ABB RobotStudio station: palet.rspag

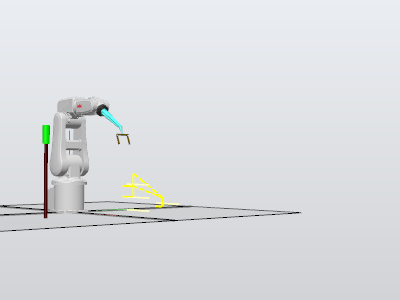
--- station ---
Station palet (saved by RobotStudio 25.3.11371.0)
Controller IRB120_3_58
  mechanical unit ROB_1: IRB120_3_58__01, 6 joints, base frame (0, 0, 0) mm
Layout (positions relative to the parent item):
  - IRB120_3_58__01 [mechanism, from %ABB.RobotStudio.Models.IRB120%\IRB120_3_58_G_01.rslib] at (0, 0, 0) mm; joint values [0, 0, 0, 0, 0.5236, 0] (rad or m)
  - traspalet [mechanism] at (364.35, 0, 594) mm, rotated rx 180 ry 60 rz 180 deg
      TCP traspalet at (31.79, 0, 229.64) mm, rotated rx 0 ry 38 rz 0 deg
      links: mytool3palet
  - YOGUR [smart component]
      signals: DI borra
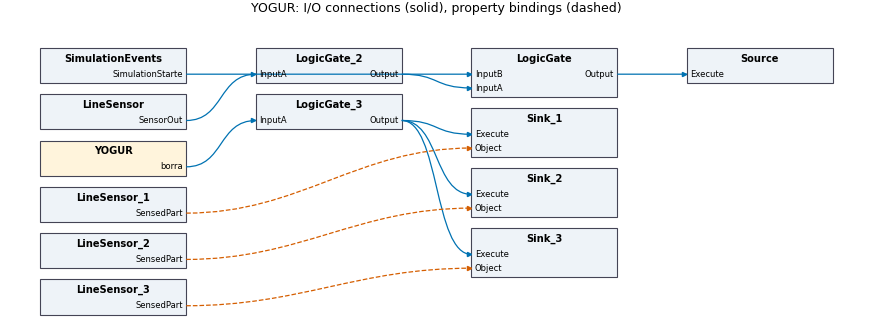
      connections:
        SimulationEvents.SimulationStarted -> LogicGate.InputB
        LogicGate.Output -> Source.Execute
        LineSensor.SensorOut -> LogicGate_2.InputA
        LogicGate_2.Output -> LogicGate.InputA
        YOGUR.borra -> LogicGate_3.InputA
        LogicGate_3.Output -> Sink_3.Execute
        LogicGate_3.Output -> Sink_2.Execute
        LogicGate_3.Output -> Sink_1.Execute
        LineSensor_1.SensedPart => Sink_1.Object
        LineSensor_2.SensedPart => Sink_2.Object
        LineSensor_3.SensedPart => Sink_3.Object
    - yogur [part] at (0, 0, 0) mm, size 60 x 80 x 72 mm
    - Source [smart component, from Components\Source.rslib]
        properties: Source=yogur; Copy=(none); Parent=(none); Position=[0.7 0.2 0]; Orientation=[0 0 0]; Transient=true; PhysicsBehavior=-1
    - SimulationEvents [smart component, from Components\SimulationEvents.rslib]
    - LogicGate [smart component, from Components\LogicGate.rslib]
        properties: Operator=OR; Delay=0
    - LineSensor [smart component, from Components\LineSensor.rslib]
        properties: Start=[0.6 0.2 0.07]; End=[0.8 0.2 0.07]; Length=0.2; Radius=0; Tag=(none); SenseMultiple=false; SensedPart=(none); SensedPoint=[0.67 0.2 0.07]
      - _sensorPart_ [part], size 200 x 0 x 0 mm
    - LogicGate_2 [smart component, from Components\LogicGate.rslib]
        properties: Operator=NOT; Delay=1
    - LineSensor_1 [smart component, from Components\LineSensor.rslib]
        properties: Start=[0.6 -0.01 0.04]; End=[0.8 -0.01 0.04]; Length=0.2; Radius=0; Tag=(none); SenseMultiple=false; SensedPart=(none); SensedPoint=[0.675910827636719 -0.00999999904632568 0.0400000038146973]
      - _sensorPart_ [part], size 200 x 0 x 0 mm
    - LineSensor_2 [smart component, from Components\LineSensor.rslib]
        properties: Start=[0.6 -0.01 0.11]; End=[0.8 -0.01 0.11]; Length=0.2; Radius=0; Tag=(none); SenseMultiple=false; SensedPart=(none); SensedPoint=[0.675313598632812 -0.01 0.11]
      - _sensorPart_ [part], size 200 x 0 x 0 mm
    - LineSensor_3 [smart component, from Components\LineSensor.rslib]
        properties: Start=[0.6 -0.01 0.18]; End=[0.8 -0.01 0.18]; Length=0.2; Radius=0; Tag=(none); SenseMultiple=false; SensedPart=(none); SensedPoint=[0 0 0]
      - _sensorPart_ [part], size 200 x 0 x 0 mm
    - Sink_1 [smart component, from Components\Sink.rslib]
        properties: Object=(none)
    - Sink_3 [smart component, from Components\Sink.rslib]
        properties: Object=(none)
    - Sink_2 [smart component, from Components\Sink.rslib]
        properties: Object=(none)
    - LogicGate_3 [smart component, from Components\LogicGate.rslib]
        properties: Operator=NOT; Delay=0
  - BALIZA [smart component]
      signals: DI COLOR
      connections:
        BALIZA.COLOR -> Highlighter.Active
    - BALIZA [part] at (400, -400, 0) mm, size 40 x 39.9 x 100 mm
    - Highlighter [smart component, from Components\Highlighter.rslib]
        properties: Object=BALIZA; Color=[255 0 0]; Opacity=255
  - SOPORTE [part] at (400, -400, 0) mm, size 20 x 20 x 400 mm
Attachment: traspalet is attached to IRB120_3_58__01 / Link6
Station logic (signal -> signal, property => property):
  IRB120_3_58.DO_0 -> BALIZA.COLOR
  IRB120_3_58.DO_0 -> YOGUR.borra

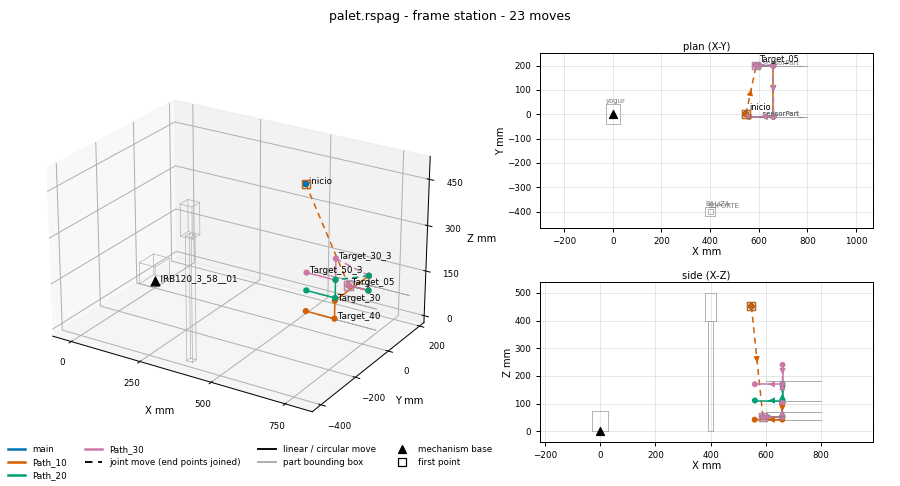
[picture p0: tool path of palet.rspag in frame station, 23 of 23 moves have a stored position in this frame; points joined in program order, loops and branches not executed]
--- Controller Data/IRB120_3_58/RAPID/TASK1/PROGMOD/CalibData.mod ---
MODULE CalibData
    PERS tooldata traspalet:=[TRUE,[[31.79,0,229.64],[0.945519,0,0.325568,0]],[1,[0,0,1],[1,0,0,0],0,0,0]];
    TASK PERS wobjdata Workobject_1:=[FALSE,TRUE,"",[[100,0,0],[1,0,0,0]],[[0,0,0],[1,0,0,0]]];
ENDMODULE

--- Controller Data/IRB120_3_58/RAPID/TASK1/PROGMOD/Module1.mod ---
MODULE Module1
    CONST robtarget Target_05:=[[489.122888793,200.000004715,51.710166889],[0.000000028,0.707106418,-0.000000043,0.707107144],[0,0,1,1],[9E+09,9E+09,9E+09,9E+09,9E+09,9E+09]];
    CONST robtarget Target_10:=[[559.122905088,199.99999557,51.710475918],[0.000000019,0.707106781,-0.000000019,0.707106781],[0,0,1,1],[9E+09,9E+09,9E+09,9E+09,9E+09,9E+09]];
    CONST robtarget Target_20:=[[559.122908398,200.000001062,101.710134289],[0.000000021,0.707106367,0.000000517,0.707107195],[0,0,1,1],[9E+09,9E+09,9E+09,9E+09,9E+09,9E+09]];
    CONST robtarget Target_30:=[[559.122903312,-10.0000012,101.709931239],[0.000000007,0.707106369,0.000000377,0.707107193],[-1,-1,2,1],[9E+09,9E+09,9E+09,9E+09,9E+09,9E+09]];
    CONST robtarget Target_40:=[[559.122925877,-9.999998556,41.709685469],[0.000000001,0.707106335,0.000000421,0.707107227],[-1,-1,2,1],[9E+09,9E+09,9E+09,9E+09,9E+09,9E+09]];
    CONST robtarget Target_50:=[[459.122816742,-9.999987978,41.709221174],[-0.000000013,0.707106336,0.000000506,0.707107226],[-1,-1,1,1],[9E+09,9E+09,9E+09,9E+09,9E+09,9E+09]];
    CONST robtarget inicio:=[[547.332902798,0,451.649052414],[0.190808996,0,0.981627183,0],[0,0,0,0],[9E+09,9E+09,9E+09,9E+09,9E+09,9E+09]];
    CONST robtarget Target_30_2:=[[560,-10,171],[0.000000007,0.707106369,0.000000377,0.707107193],[-1,-1,2,1],[9E+09,9E+09,9E+09,9E+09,9E+09,9E+09]];
      CONST robtarget Target_30_3:=[[560,-10,240],[0.000000007,0.707106369,0.000000377,0.707107193],[-1,-1,2,1],[9E+09,9E+09,9E+09,9E+09,9E+09,9E+09]];
    CONST robtarget Target_40_2:=[[560,-10,111],[0.000000001,0.707106335,0.000000421,0.707107227],[-1,-1,2,1],[9E+09,9E+09,9E+09,9E+09,9E+09,9E+09]];
     CONST robtarget Target_40_3:=[[560,-10,170],[0.000000001,0.707106335,0.000000421,0.707107227],[-1,-1,2,1],[9E+09,9E+09,9E+09,9E+09,9E+09,9E+09]];
    CONST robtarget Target_50_2:=[[460,-10,111],[-0.000000013,0.707106336,0.000000506,0.707107226],[-1,-1,2,1],[9E+09,9E+09,9E+09,9E+09,9E+09,9E+09]];
     CONST robtarget Target_50_3:=[[460,-10,170],[-0.000000013,0.707106336,0.000000506,0.707107226],[-1,-1,2,1],[9E+09,9E+09,9E+09,9E+09,9E+09,9E+09]];
    VAR num cajas;
    !***********************************************************
    !

    !***********************************************************
    PROC main()
          TPErase;
        RESET DO_0;
        TPWrite "Escribre entre 1 y 3, ";
      TPReadNum cajas, "el número de yogures que quieres apilar";
      TPErase;

        TPErase;
      IF cajas<1 OR cajas>3 THEN
             TPWrite "";
          TPWrite "EL NÚMERO INTRODUCIDO NO ESTA ENTRE 1 Y 3 VUELVE A INTENTARLO";
          WaitTime 3;
          TPErase;
      ELSE
           TPWrite "VAS A COLOCAR ";
          TPWrite ""\Num:=cajas;
            TPWrite "YOGURES ";
        WaitTime 3;
          Set DO_0;
          MoveJ inicio,v200,z100,traspalet\WObj:=wobj0;
       TEST cajas
       CASE 1:

            Path_10;
            MoveJ inicio,v200,z100,traspalet\WObj:=wobj0;
       CASE 2:

            Path_10;
            Path_20;
            MoveJ inicio,v200,z100,traspalet\WObj:=wobj0;
      CASE 3:
            Path_10;
            Path_20;
             Path_30;
             MoveJ inicio,v200,z100,traspalet\WObj:=wobj0;
       ENDTEST
      ENDIF
    ENDPROC
    PROC Path_10()
        MoveJ inicio,v200,z100,traspalet\WObj:=wobj0;
        MoveJ Target_05,v200,z100,traspalet\WObj:=Workobject_1;
        MoveL Target_10,v200,z100,traspalet\WObj:=Workobject_1;
        MoveL Target_20,v200,z0,traspalet\WObj:=Workobject_1;
        MoveL Target_30,v200,z100,traspalet\WObj:=Workobject_1;
        MoveL Target_40,v200,z0,traspalet\WObj:=Workobject_1;
        MoveL Target_50,v200,z100,traspalet\WObj:=Workobject_1;


    ENDPROC
      PROC Path_20()


        MoveL Target_05,v200,z100,traspalet\WObj:=Workobject_1;
        MoveL Target_10,v200,z100,traspalet\WObj:=Workobject_1;
        MoveL Target_20,v200,z100,traspalet\WObj:=Workobject_1;
        MoveJ Target_30_2,v200,z100,traspalet\WObj:=Workobject_1;
        MoveL Target_40_2,v200,z0,traspalet\WObj:=Workobject_1;
        MoveL Target_50_2,v200,z100,traspalet\WObj:=Workobject_1;

    ENDPROC
      PROC Path_30()

        MoveL Target_05,v200,z100,traspalet\WObj:=Workobject_1;
        MoveL Target_10,v200,z100,traspalet\WObj:=Workobject_1;
        MoveL Target_20,v200,z100,traspalet\WObj:=Workobject_1;
        MoveJ Target_30_3,v200,z100,traspalet\WObj:=Workobject_1; !COLOCADO
        MoveL Target_40_3,v200,z0,traspalet\WObj:=Workobject_1;  !BAJO
        MoveL Target_50_3,v200,z100,traspalet\WObj:=Workobject_1; ! ME RETIRO

    ENDPROC
ENDMODULE

--- Controller Data/IRB120_3_58/SYSPAR/EIO.cfg ---
EIO:CFG_1.0:6:1::
#
INDUSTRIAL_NETWORK:

      -Name "DeviceNet" -Label "DeviceNet Master/Slave Network" -Address "2"
#
DEVICENET_DEVICE:

      -Name "d652" -VendorName "ABB Robotics" -ProductName "24 VDC I/O Device"\
      -Label "DSQC 652 24 VDC I/O Device" -Address 10 -ProductCode 26\
      -DeviceType 7 -ConnectionType "COS" -OutputSize 2 -InputSize 2
#
DEVICENET_INTERNAL_DEVICE:

      -Name "DN_Internal_Device" -VendorName "ABB Robotics"\
      -ProductName "DeviceNet Internal Slave Device"
#
EIO_SIGNAL:

      -Name "DI_0" -SignalType "DI" -Device "d652" -DeviceMap "0" -Access "All"

      -Name "DO_0" -SignalType "DO" -Device "d652" -DeviceMap "0" -Access "All"

      -Name "DI_1" -SignalType "DI" -Device "d652" -DeviceMap "1" -Access "All"

      -Name "DI_2" -SignalType "DI" -Device "d652" -DeviceMap "2" -Access "All"

      -Name "DI_3" -SignalType "DI" -Device "d652" -DeviceMap "3" -Access "All"

      -Name "DI_4" -SignalType "DI" -Device "d652" -DeviceMap "4" -Access "All"

      -Name "DI_5" -SignalType "DI" -Device "d652" -DeviceMap "5" -Access "All"

      -Name "DO_1" -SignalType "DO" -Device "d652" -DeviceMap "1" -Access "All"

      -Name "DO_2" -SignalType "DO" -Device "d652" -DeviceMap "2" -Access "All"

      -Name "DO_3" -SignalType "DO" -Device "d652" -DeviceMap "3" -Access "All"

      -Name "DO_4" -SignalType "DO" -Device "d652" -DeviceMap "4" -Access "All"

      -Name "DO_5" -SignalType "DO" -Device "d652" -DeviceMap "5" -Access "All"
